FUNCTION_BLOCK SC_PostPalletizer EXTENDS FB_Chain
VAR_INPUT
	bExecute : BOOL;
	bPalletizerDeliveryRequest : BOOL;
	sTLMqttName : STRING(8);
END_VAR
VAR_OUTPUT
	bGrantDeliveryPermission : BOOL;
END_VAR
VAR
	
	fbPalletAvailable : Sensor;
	fbRollConveyor : RollerConveyor;
	
END_VAR

SUPER^();
fbPalletAvailable();
fbRollConveyor();

METHOD PROTECTED   Busy : BOOL
VAR_INPUT
END_VAR
VAR
	stMqttPayload : ST_MqttPayload;
	messageIndex : UINT;
END_VAR
fbStepWorkerBusy();
CASE fbStepWorkerBusy.uiStep OF
	
	0: 
		THIS^.fbRollConveyor.On();
		rChainController.releaseForChain('scFirstFloor', THIS^);
		fbStepWorkerBusy.mNextStep(10);
		
	10:
		IF THIS^.fbPalletAvailable.bSignal
		THEN
			THIS^.fbRollConveyor.Off();
			fbStepWorkerBusy.mNextStep(20);
		END_IF
	
	20: 
		
		//Mqtt exchange
		IF Ads.fbMqttClient.Publish(sTLMqttName,stMqttPayload)
		THEN
			fbStepWorkerBusy.mNextStep(30);
		END_IF
	
	30:
	
		messageIndex := ADS.fbMqttClient.isNewMessage(sTLMqttName);
		IF messageIndex > 0
		THEN
			stMqttPayload := Ads.fbMqttClient.getNewMessage(messageIndex);
			fbStepWorkerBusy.mNextStep(40);
		END_IF
		
	40:
	
		THIS^.fbRollConveyor.On();
		fbStepWorkerBusy
			.mSetTimer(T#2S)
			.mNextStep(50);
			
	50:
		
		THIS^.fbRollConveyor.Off();
		Done();
		fbStepWorkerBusy.mNextStep(0);
		
END_CASE
END_METHOD

METHOD PROTECTED  Error : BOOL
VAR_INPUT
END_VAR
END_METHOD

METHOD PROTECTED  Idle : BOOL
VAR_INPUT
END_VAR
END_METHOD

METHOD PROTECTED  Init : BOOL
VAR_INPUT
END_VAR
IF ADS.fbMqttClient.Subscribe(sTopic := sTLMqttName)
THEN			
	Start();
END_IF
END_METHOD

METHOD PROTECTED  Prepare : BOOL
VAR_INPUT
END_VAR
END_METHOD

METHOD PROTECTED  Ready : BOOL
VAR_INPUT
END_VAR

fbStepWorkerReady();
CASE fbStepWorkerReady.uiStep OF
	
0:

	IF bExecute
		AND NOT fbPalletAvailable.bSignal
	THEN
		fbStepWorkerReady.mNextStep(10);
	END_IF
		
10:
	IF rChainController
		.releaseCheck(THIS^)
		.releaseFromChain(sChainReleasing := 'scFirstFloor', THIS^)
		.releaseResult(THIS^) 
	THEN
		fbStepWorkerReady.mNextStep(0);
		Execute();
	END_IF
	
END_CASE
END_METHOD

METHOD PROTECTED  Waiting : BOOL
VAR_INPUT
END_VAR
END_METHOD

END_FUNCTION_BLOCK

(* stored: Version 1.1.0.1, ProductVersion 3.1.4024.2
   POU SC_PostPalletizer: Id {85befc7a-2bdd-4f2e-96bb-ac167a701ce0}, SpecialFunc None
   Method Busy: Id {2bd66645-72ae-4316-97cd-fa00de023996}
   Method Error: Id {1cc12c3d-3d64-4bd9-b820-a691065cd20e}
   Method Idle: Id {21e079be-ae67-4053-80ab-63c89c0c93d1}
   Method Init: Id {43dca436-b609-4d32-a22f-f3731cf758bf}
   Method Prepare: Id {80d62777-b07d-4ce4-9d67-fe49f794d2f0}
   Method Ready: Id {8a8fa7c7-11ba-4410-a809-27bdd057d24c}
   Method Waiting: Id {a61fe33e-cd23-4d8a-8570-78b7878b4290} *)
